FUNCTION_BLOCK F_DIV (* Divides two values *)
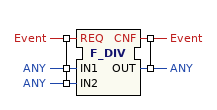
  EVENT_INPUT
    REQ WITH IN1, IN2; (* Normal Execution Request *)
  END_EVENT
  EVENT_OUTPUT
    CNF WITH OUT; (* Execution Confirmation *)
  END_EVENT
  VAR_INPUT
    IN1 : ANY; (* First funtion input *)
    IN2 : ANY; (* Second function input *)
  END_VAR
  VAR_OUTPUT
    OUT : ANY; (* Function output *)
  END_VAR
END_FUNCTION_BLOCK
